INTERFACE Disposable EXTENDS __System.IQueryInterface

METHOD PUBLIC Dispose
END_METHOD

END_INTERFACE

(* stored: Version 1.1.0.1
   Itf Disposable: Id {0ac8ea4a-8a07-4e17-87b2-50ddcba07e56}
   Method Dispose: Id {860d07a8-49bb-4a9d-a729-17f246fb69b8} *)
